// This function has been automatically generated from the project information.
{attribute 'signature_flag' := '1073741824'}
{attribute 'TcGenerated'}
{attribute 'no-analysis'}
FUNCTION F_GetCompany : WSTRING
VAR_INPUT
	
END_VAR

F_GetCompany := "Beckhoff UK";

END_FUNCTION

(* stored: Version 1.1.0.1
   POU F_GetCompany: Id {db7aa69a-10b2-45c3-a512-0b9eb2481fc4}, SpecialFunc None *)
